FUNCTION StateEnabled : BOOL
VAR_INPUT
END_VAR
VAR
END_VAR

END_FUNCTION

(* stored: Version 1.1.0.1, ProductVersion 3.1.4022.18
   POU StateEnabled: Id {37de7ef5-3890-457b-b3b9-3d3f0accca78}, SpecialFunc None *)
